# B&R Automation Studio project mappMotion
Automation Studio 4.5.3.86 SP; technology packages: mappCockpit 5.8.0, mappMotion 5.8.0, mappView 5.8.0

## Configuration Config1

CPU X20CP3585, AutomationRuntime D4.52, Build 4.1.2, Vc V4.52.0

### Task classes (Cpu.sw)
```
Cyclic#1:
  Program <- Program.prg
DataObjects: McAcpSys
Binaries: arsvcreg, udbdef, mvLoader, McAcpDrv, arflatprv, McProfGen, arcoal, TCData, mCoWebSc, McAcpSim, Role, Config_2, iomap, arconfig, asfw, sysconf, User, Settings, ashwac, Config_1, ashwd
Libraries: McBase, MpAxis, McAxis, MpBase, CoTrace, AsZip, FileIO, runtime, McDS402Ax, McPureVAx, asieccon, powerlnk, astime, sys_lib, asepl
```

### Hardware
```
8I76xxxxxxx.0P-xxx : 8I76xxxxxxx.0P-xxx v1.1.0.5  [PLK1 -> X20CP3585.IF3 (NodeNumber=5) [Cable Type=PowerlinkCable, Length=10, Version=1.0.0.2]]
  FunctionModel = MotionConfig
  Supervision = off
  McTypeID = McAcoposInverterP76P
  AxisReference = gAxis_Inv
  InputIsReadOnly = 0
  Input = 1
  OutputIsReadOnly = 0
  Output = 1
  ReferenceDistanceIsReadOnly = 0
  ReferenceDistance = 1
  UnitOfSetpoint = Rpm
  IOM_AIDP1 = LFT
  Sel_NameplateMask = 8Ix6S200037_IEC
  Cfg_NSP = 880
  Cfg_NCR = 18
  Cfg_COS = 100
  Cfg_NPR = 18
  Cfg_TUNU = 0
  Sel_DCtype = 8Ix6S2V240_FIX
  Cfg_SPG = 20
X20CP3585 : X20CP3585 v1.6.0.0
  Connector IF2:
    ActivateDevice = 1
    Mode = Manual
    InternetAddress = 192.168.0.34
    SubnetMask = 255.255.255.0
  ConfigurationID = mappMotion_Config1
  FileDevice1
  FileDeviceName1 = USER
  FileDevicePath1 = F:\
  ActivateOpcUa = 1
  OpcUa_AuthenticationSecurityPolicy_EnableNone = 1
  OpcUa_AuthenticationSecurityPolicy_EnableBasic128Rsa15 = 1
  OpcUaInformationModels_PV_Version = 1
```

### Config_1.axis - X20CP3585/mappMotion/Config_1.axis
```
Element gAxis_Inv (Type=axis)
  BaseTypeIsReadOnly = 0
  BaseType = Rotary
    MeasurementUnitIsReadOnly = 0
    MeasurementUnit = 17476
    MeasurementResolutionIsReadOnly = 0
    MeasurementResolution = 1
    CountDirectionIsReadOnly = 0
    CountDirection = Standard
  MovementLimitsIsReadOnly = 0
  MovementLimits = Internal
    Position:
      LowerLimitMin = -1.79769313486231E308
      UpperLimitMax = 1.79769313486231E308
      LowerLimit = -10000.0
      UpperLimit = 10000.0
    VelocityIsReadOnly = 0
    Velocity:
      VelocityMax = 3.4E38
      Velocity = 5280
    AccelerationIsReadOnly = 0
    Acceleration:
      AccelerationMax = 3.4E38
      Acceleration = 1e6
    DecelerationIsReadOnly = 0
    Deceleration:
      DecelerationMax = 3.4E38
      Deceleration = 1e6
  Alarms = None
Element gVAxis_Inv (Type=axis)
  BaseTypeIsReadOnly = 0
  BaseType = LinearBounded
    MeasurementUnit = 5066068
    MeasurementResolutionIsReadOnly = 0
    MeasurementResolution = 0.1
    CountDirectionIsReadOnly = 0
    CountDirection = Standard
  MovementLimitsIsReadOnly = 0
  MovementLimits = Internal
    Position:
      LowerLimitMin = -1.79769313486231E308
      UpperLimitMax = 1.79769313486231E308
      LowerLimit = -1000.0
      UpperLimit = 1000.0
    VelocityIsReadOnly = 0
    Velocity:
      VelocityMax = 3.4E38
      Velocity = 146
    AccelerationIsReadOnly = 0
    Acceleration:
      AccelerationMax = 3.4E38
      Acceleration = 500
    DecelerationIsReadOnly = 0
    Deceleration:
      DecelerationMax = 3.4E38
      Deceleration = 500
  Alarms = None
```

### Config_2.purevaxcfg - X20CP3585/mappMotion/Config_2.purevaxcfg
```
Element gPureVirtualAxis_Inv (Type=purevaxcfg)
  TypeID = PureVAxConfig
  PureVAxis:
    AxisReference = gVAxis_Inv
    Homing:
      Mode = Direct
        Position = 0.0
    JerkFilter = NotUsed
```

## Logical view

Binary libraries used (declarations not repeated): operator, runtime, astime, AsIecCon, McBase 5.08.0, MpAxis 5.08.0, McAxis 5.08.0, MpBase 5.08.0, CoTrace 5.08.0, AsZip, FileIO, McDS402Ax 5.08.0, McPureVAx 5.08.0


### Program Logical/Program (IEC)

#### Cyclic.st - Cyclic code
```iecst
PROGRAM _CYCLIC

	MpAxisBasic_0(
		Stop := MC_ReadStatus_0.ErrorStop
	);

	MC_Power_0(
		Enable := MpAxisBasic_0.PowerOn
	);

	MC_BR_VelocityControl_0(
		Enable := MC_Power_0.Status,
		CyclicVelocity := MpAxisBasic_0.Velocity / 10 * 360
	);

	MC_ReadStatus_0();

	MC_ReadActualVelocity_0();
	Position := Position + MC_ReadActualVelocity_0.Velocity * 0.01;

	MC_Reset_0();
END_PROGRAM
```

#### Init.st - Init code
```iecst
PROGRAM _INIT
	MpAxisBasic_0(
		MpLink := ADR(gVAxis_Inv),
		Enable := FALSE ,
		Parameters := ADR(MpAxisParameters)

	);
	MpAxisBasic_0.Enable := TRUE;

	MC_Power_0(
		Axis := ADR(gAxis_Inv),
		Enable := FALSE
	);

	MC_ReadStatus_0(
		Axis := ADR(gAxis_Inv),
		Enable := TRUE
	);

	AdvancedParameters.Acceleration := 1e6;
	AdvancedParameters.Deceleration := 1e6;
	AdvancedParameters.Jerk := 0.0;
	MC_BR_VelocityControl_0(
		Axis := ADR(gAxis_Inv),
		Enable := FALSE,
		AdvancedParameters := AdvancedParameters,
		CyclicVelocity := 0
	);

	MC_ReadActualVelocity_0(
		Axis := ADR(gAxis_Inv),
		Enable := TRUE
	);

	MC_Reset_0(
		Axis := ADR(gAxis_Inv),
		Execute := FALSE
	);

END_PROGRAM
```

#### Exit.st - Exit code
```iecst
PROGRAM _EXIT
	MC_Power_0( Enable := FALSE );
	MC_BR_VelocityControl_0( Enable := FALSE );
	MpAxisBasic_0( Enable := FALSE );

END_PROGRAM
```

#### Variables.var - Local variables
```iecst
VAR
	MpAxisParameters : MpAxisBasicParType;
	MpAxisBasic_0 : MpAxisBasic;
	MC_Power_0 : MC_Power;
	MC_Reset_0 : MC_Reset;
	AdvancedParameters : McAdvVelCtrlParType;
	MC_BR_VelocityControl_0 : MC_BR_VelocityControl;
	MC_ReadActualVelocity_0 : MC_ReadActualVelocity;
	Position : LREAL;
	MC_ReadStatus_0 : MC_ReadStatus;
END_VAR
```

Listed in the project but not available here: Logical/Global.typ, Logical/Global.var, Logical/Program/Types.typ
